// TwinCAT 3 PLC project TcUnit
// Title: TcUnit
// Company: www.tcunit.org
// Author: Jakob Sagatowski and other contributors, see CONTRIBUTORS file on www.github.com/tcunit/TcUnit
// ProjectVersion: 0.4.1.0
// Description: TwinCAT unit testing framework. Documentation and examples are available at www.tcunit.org
// ProgramVersion: 3.1.4022.2
// libraries:
//   Tc2_Standard, * (Beckhoff Automation GmbH)
//   Tc2_System, * (Beckhoff Automation GmbH)
//   Tc2_Utilities, * (Beckhoff Automation GmbH)
//   Base Interfaces,newest,System
// project tree:
//   DUTs/ E_TestSuiteRunState.TcDUT (not stored), MaxString.TcDUT, ST_AssertResult.TcDUT (not stored), TypeClass.TcDUT, U_ExpectedOrActual.TcDUT (not stored)
//   GVLs/ GVL.TcGVL (not stored), GVL_Constants.TcGVL (not stored)
//   ITFs/ I_AssertMessageFormatter.TcIO (not stored), I_RunnableTestSuite.TcIO (not stored), I_TestSuite.TcIO (not stored), I_TestResultFormatter.TcIO (not stored)
//   POUs/ FB_ADSTestResultFormatter.TcPOU (not stored), FB_AnyComparator.TcPOU (not stored), FB_Assert.TcPOU (not stored), FB_AssertResultStatic.TcPOU (not stored), FB_ADSAssertMessageFormatter.TcPOU (not stored), FB_TcUnitRunner.TcPOU (not stored), FB_Test.TcPOU (not stored), FB_TestSuite.TcPOU (not stored)
//   POUs/Functions/ F_AnyToUnionValue.TcPOU (not stored), F_AnyTypeClassToString.TcPOU (not stored), F_IsAnyEqualToUnionValue.TcPOU (not stored), F_RemoveInstancePathAndProjectNameFromTestInstancePath.TcPOU (not stored), RUN.TcPOU (not stored), TEST.TcPOU (not stored), anyToString.TcPOU
//   POUs/NewVersion/ IRunner.TcIO, ITestSuite.TcIO, UnitTest.TcPOU, UnitTestPrinter.TcPOU, UnitTestRunner.TcPOU, UnitTestSuite.TcPOU
//   POUs/StringBuilder/ SimpleStringBuilder.TcPOU
//   Version/ Global_Version.TcGVL (not stored)

// ---- DUTs/MaxString.TcDUT
TYPE MaxString : STRING(255); END_TYPE

// ---- DUTs/TypeClass.TcDUT
{attribute 'qualified_only'}
{attribute 'strict'}
TYPE TypeClass :
(
	TYPE_BOOL := 0,
  TYPE_BIT := 1,
  TYPE_BYTE := 2,
  TYPE_WORD := 3,
  TYPE_DWORD := 4,
  TYPE_LWORD := 5,
  TYPE_SINT := 6,
  TYPE_INT := 7,
  TYPE_DINT := 8,
  TYPE_LINT := 9,
  TYPE_USINT := 10,
  TYPE_UINT := 11,
  TYPE_UDINT := 12,
  TYPE_ULINT := 13,
  TYPE_REAL := 14,
  TYPE_LREAL := 15,
  TYPE_STRING := 16,
  TYPE_WSTRING := 17,
  TYPE_TIME := 18,
  TYPE_DATE := 19,
  TYPE_DATEANDTIME := 20,
  TYPE_TIMEOFDAY := 21,
  TYPE_POINTER := 22,
  TYPE_REFERENCE := 23,
  TYPE_SUBRANGE := 24,
  TYPE_ENUM := 25,
  TYPE_ARRAY := 26,
  TYPE_PARAMS := 27,
  TYPE_USERDEF := 28,
  TYPE_NONE := 29,
  TYPE_ANY := 30,
  TYPE_ANYBIT := 31,
  TYPE_ANYDATE := 32,
  TYPE_ANYINT := 33,
  TYPE_ANYNUM := 34,
  TYPE_ANYREAL := 35,
  TYPE_LAZY := 36,
  TYPE_LTIME := 37,
  TYPE_BITCONST := 38,
  TYPE_INTERFACE := 16#F000
);
END_TYPE

// ---- POUs/NewVersion/IRunner.TcIO
INTERFACE IRunner

METHOD registerTestSuite
VAR_INPUT
    testSuite: ITestSuite;
END_VAR
END_METHOD

END_INTERFACE

// ---- POUs/NewVersion/ITestSuite.TcIO
INTERFACE ITestSuite

METHOD runAllTests
VAR_INPUT
END_VAR
END_METHOD

END_INTERFACE

// ---- POUs/Functions/anyToString.TcPOU
FUNCTION anyToString : MaxString
VAR_INPUT
  toTransform: ANY;
END_VAR
VAR
  intPtr: POINTER TO INT;
  realPtr: POINTER TO REAL;
  stringPtr: POINTER TO STRING;
END_VAR

CASE UDINT_TO_INT(toTransform.TypeClass) OF
TypeClass.TYPE_INT:
  intPtr := toTransform.pValue;
  anyToString := TO_STRING(intPtr^);
TypeClass.TYPE_REAL:
  realPtr := toTransform.pValue;
  anyToString := TO_STRING(realPtr^);
TypeClass.TYPE_STRING:
  stringPtr := toTransform.pValue;
  anyToString := stringPtr^;
ELSE
  anyToString := '';
END_CASE

END_FUNCTION

// ---- POUs/NewVersion/UnitTest.TcPOU
FUNCTION_BLOCK UnitTest
VAR_INPUT
END_VAR
VAR_OUTPUT
END_VAR
VAR
    _testSuite: ITestSuite;
END_VAR

METHOD FB_init : BOOL
VAR_INPUT
	bInitRetains : BOOL; // if TRUE, the retain variables are initialized (warm start / cold start)
	bInCopyCode : BOOL;  // if TRUE, the instance afterwards gets moved into the copy code (online change)
    _testSuite: ITestSuite;
END_VAR
THIS^._testSuite := _testSuite;
END_METHOD

PROPERTY testSuite : ITestSuite
GET
testSuite := THIS^._testSuite;
END_GET
SET
END_SET
END_PROPERTY

END_FUNCTION_BLOCK

// ---- POUs/NewVersion/UnitTestPrinter.TcPOU
FUNCTION_BLOCK UnitTestPrinter
VAR_INPUT
END_VAR
VAR_OUTPUT
END_VAR
VAR
    messageBuilder: SimpleStringBuilder;
END_VAR

METHOD getFailureMessage : MaxString
VAR_INPUT
    expected: ANY;
    actual: ANY;
    message: MaxString;
    path: MaxString;
END_VAR
VAR
    messageToAppend: MaxString;
END_VAR
messageToAppend := 'FAILED TEST $'';
messageBuilder.append(messageToAppend);
messageBuilder.append(path);
messageToAppend := '$', EXP: ';
messageBuilder.append(messageToAppend);
messageBuilder.append(expected);
messageToAppend := ', ACT: ';
messageBuilder.append(messageToAppend);
messageBuilder.append(actual);
messageToAppend := ', MSG: ';
messageBuilder.append(messageToAppend);
messageBuilder.append(message);

getFailureMessage := messageBuilder.toString();
END_METHOD

METHOD printFailure
VAR_INPUT
    expected: MaxString;
    actual: MaxString;
    message: MaxString;
    path: MaxString;
END_VAR
VAR
    failureMessage: MaxString;
END_VAR
failureMessage := getFailureMessage(expected, actual, message, path);
END_METHOD

END_FUNCTION_BLOCK

// ---- POUs/StringBuilder/SimpleStringBuilder.TcPOU
FUNCTION_BLOCK SimpleStringBuilder
VAR_INPUT
END_VAR
VAR_OUTPUT
END_VAR
VAR
    builderString: MaxString;
END_VAR

METHOD append
VAR_INPUT
    toAppend: ANY;
END_VAR
VAR
    strToAppend: MaxString;
END_VAR
strToAppend := anyToString(toAppend);
builderString := CONCAT(builderString, strToAppend);
END_METHOD

METHOD toString : MaxString
toString := builderString;
END_METHOD

END_FUNCTION_BLOCK

// ---- POUs/NewVersion/UnitTestRunner.TcPOU
FUNCTION_BLOCK UnitTestRunner IMPLEMENTS IRunner
VAR_INPUT
END_VAR
VAR_OUTPUT
END_VAR
VAR
    testSuites: ARRAY [0..10] OF ITestSuite;
END_VAR

PROPERTY numberOfTestSuites : UINT
GET
VAR
    i: INT;
END_VAR
numberOfTestSuites := 0;
FOR i:=0 TO 10 DO
    IF THIS^.testSuites[i] <> 0 THEN
        numberOfTestSuites := numberOfTestSuites + 1;
    ELSE
        EXIT;
	END_IF
END_FOR
END_GET
END_PROPERTY

METHOD registerTestSuite
VAR_INPUT
    testSuite: ITestSuite;
END_VAR
VAR
    i: INT;
END_VAR
FOR i:=0 TO 10 DO
    IF THIS^.testSuites[i] = testSuite THEN
        EXIT;
	END_IF
    IF THIS^.testSuites[i] = 0 THEN
        THIS^.testSuites[i] := testSuite;
        EXIT;
	END_IF
END_FOR
END_METHOD

METHOD runAllTests
VAR
    i: INT;
END_VAR
FOR i:=0 TO 10 DO
    IF testSuites[i] = 0 THEN
        EXIT;
	END_IF
    testSuites[i].runAllTests();
END_FOR
END_METHOD

END_FUNCTION_BLOCK

// ---- POUs/NewVersion/UnitTestSuite.TcPOU
FUNCTION_BLOCK UnitTestSuite IMPLEMENTS ITestSuite
VAR_INPUT
END_VAR
VAR_OUTPUT
END_VAR
VAR
END_VAR

METHOD FB_init : BOOL
VAR_INPUT
	bInitRetains : BOOL; // if TRUE, the retain variables are initialized (warm start / cold start)
	bInCopyCode : BOOL;  // if TRUE, the instance afterwards gets moved into the copy code (online change)
    runner: IRunner;
END_VAR
IF runner <> 0 THEN
    runner.registerTestSuite(THIS^);
END_IF
END_METHOD

PROPERTY numberOfTests : UINT
GET
END_GET
END_PROPERTY

{warning 'add method implementation'}
METHOD runAllTests
END_METHOD

END_FUNCTION_BLOCK
